FUNCTION_BLOCK servo

VAR_INPUT
	
offline_bit: BOOL;
error_bit: BOOL	;
servo_absolute: BOOL;
target_position: REAL;
servo_pos_delay_time: LTIME;
END_VAR

VAR_OUTPUT
	servo_pos_delay_time_display: LTIME;
	actual_position: REAL;
	absolute_done: BOOL;
END_VAR

VAR
	delay : lton;
	
END_VAR

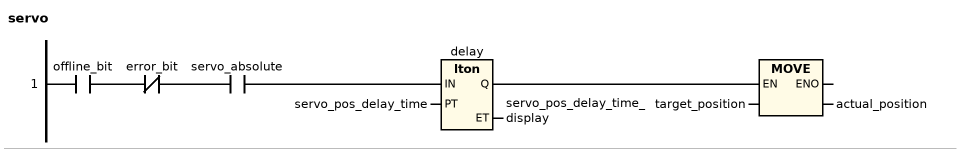
// NETWORK 1
delay(
    IN := offline_bit AND NOT error_bit AND servo_absolute,
    PT := servo_pos_delay_time,
    ET => servo_pos_delay_time_display); // lton
IF delay.Q THEN actual_position := target_position; END_IF

END_FUNCTION_BLOCK

(* stored: Version 1.1.0.1, ProductVersion 3.1.4024.11
   POU servo: Id {083be752-38d7-497e-a40b-17d29634cc94}, SpecialFunc None *)
